// TIA Portal V20 export
FUNCTION_BLOCK "FB_BrakeTest"   // FB412, SCL
TITLE = BrakeTest
{ S7_Optimized_Access := 'FALSE' }
VERSION : 3.12
// Sinamics brake test
// stored: AutoNumber false, IsIECCheckEnabled true, SetENOAutomatically false
   VAR_INPUT
      iStartBt : Bool;   // start BT (Bit must only be resetted as soon as done = 1)
      iQuit : Bool;   // quit error
      iExternalBrakeClosed : Bool;   // feedback external brake; if closed = 1, if open = 0
      iMaxStepTime : Time := T#6S;   // max time per sequencer step
      iBrakeNum : Bool;   // number of brake to be tested; brake 1 = 0; brake 2 = 1
      iActivateAutoDirection : Bool;   // enable automatic detection of direction of test torque
      iSetManualDirection : Bool;   // manual selection of direction of test torque
      iTestSequence : Bool;   // selection of test sequence; sequence 1 = 0, sequence 2 = 1
   END_VAR
   VAR_OUTPUT
      oCloseExternalBrake : Bool;   // signal to close the external brake; close = 1, open = 0
      oDone : Bool;   // done without errors
      oError : Bool;   // error occurred
      oStateNum : Int;   // active step of the sequence
      oDiagnoseError : Int;   // error number
      oError1 : Bool;   // invalid sequence step
      oError2 : Bool;   // invalid start condition: axis not stationery
      oError3 : Bool;   // invalid start condition: pulse enable missing
      oError4 : Bool;   // brake test noch successful
      oError5 : Bool;   // sequence step time monitoring error
      oError6 : Bool;   // startBT reset while in progress
      oError7 : Bool;   // invalid error number
      oError8 : Bool;   // no feedback external brake within "maxStepTime"
   END_VAR
   VAR_IN_OUT
      ioAxisDB : "LBP_typeAxisX";   // UDT of test axis (has to be connected!)
   END_VAR
   VAR
      sStepNum : Int;   // active sequencer step
      sEdgeFlagStop : Bool;   // falling edge flag of startBT
      sEdgeFlagStart : Bool;   // rising edge flag of startBT
      sStepNumOld : Int;   // sequencer step of the previous PLC cycle
      sBTDeselectionDelay : Bool;   // TOF, Q output of deselection timer
      sStartTimer { ExternalVisible := 'False'; ExternalWritable := 'False'} : Bool := true;   // start timer of sequencer time monitoring
      sActiveError : Bool;   // active error
      sInstIecTimerTimeStepBt { S7_SetPoint := 'True'} : TOF_TIME;   // timer for monitoring the steps of the sequencer
      sInstIecTimerSelectSafeBt { S7_SetPoint := 'True'} : TOF_TIME;   // timer to delay the program, if BT is deselected
      sErrorNum { ExternalVisible := 'False'; ExternalWritable := 'False'} : Int;   // provisional error number
   END_VAR
   VAR_TEMP
      tIncrement : Bool;   // increment sequencer
      tTimeSig : Bool;   // TOF, Q output sequencer time monitoring
      tRisBTStart : Bool;   // rising edge startBT
      tFalBTStart : Bool;   // falling edge startBT
      tErr6 : Bool;   // error no. 6
   END_VAR
BEGIN
   REGION BLOCK INFO HEADER
   //=============================================================================
   // Siemens
   // (c)Copyright 2021 All Rights Reserved
   // ----------------------------------------------------------------------------
   // Library:       Lib_SBT_SINUMERIK_ONE
   // Tested with:   V6.13 / NCU 1760
   // Engineering:   TIA Portal V16 Update 4
   // Restrictions:  -
   // Requirements:  motor with brake; UDT "LBP_typeAxisX" of the axis to be tested
   // Functionality: brake test for safety axis
   // ----------------------------------------------------------------------------
   // Change log table:
   // Version   Date         Expert in charge   Changes applied
   // 03.01.02  01.12.2021   Siemens AG         First released version
   // =============================================================================
   END_REGION BLOCK INFO HEADER

   REGION set temp variables 
     #tErr6 := 0;
     #tIncrement := 0;
     #tTimeSig := 0;
     #tRisBTStart := 0;
     #tFalBTStart := 0;
   END_REGION

   REGION edge evaluation 
     // rising edge startBt 
     #tRisBTStart := (#iStartBt AND NOT #iQuit) AND NOT #sEdgeFlagStart;
     #sEdgeFlagStart := (#iStartBt AND NOT #iQuit);

     // falling edge startBt 
     #tFalBTStart := NOT #iStartBt AND #sEdgeFlagStop;
     #sEdgeFlagStop := #iStartBt;
   END_REGION

   REGION return function if Test is inactive 
     // return function while Test is inactive 
     IF NOT (#iStartBt OR #tFalBTStart OR #tRisBTStart OR
       #sActiveError OR #iQuit) THEN
       RETURN;
   END_IF;
   END_REGION

   REGION reset brake test enable when FB stopped 
     IF NOT (#iStartBt OR #sActiveError) THEN
       IF #sStepNum <> 0 THEN
         //error number 6: SBT is cancelled with startBt=0 
         #tErr6 := 1;
       END_IF;
       //stop step sequence 
       #sStepNum := 0;
       //Cancellation/deselection SBT 
       #ioAxisDB.A_StartBrakeTest := 0;
       #ioAxisDB.SCC.CW3.SelectionSBT := 0;
       #ioAxisDB.SCC.CW3.BT_Start := 0;
     END_IF;
   END_REGION

   REGION external brake status/control 
     IF #iStartBt THEN
       //control external brake 
       #oCloseExternalBrake := #ioAxisDB.SIC.SW3.BrakeReq;
       //status external brake 
       #ioAxisDB.SCC.CW3.BrakeClosed := #iExternalBrakeClosed;
     END_IF;

   END_REGION

   REGION timer 
     //start Watchdog Timer on the beginning and for every new step 
     #sStartTimer := 0;
     IF (#sStepNum <> #sStepNumOld)
       OR (#tRisBTStart = 1) THEN
       #sStartTimer := 1;
     END_IF;

     // Timer (TOF) Time delay stop SBT 
     #sInstIecTimerSelectSafeBt(IN := #ioAxisDB.A_StartBrakeTest,
                               PT := T#100ms,
                               Q => #sBTDeselectionDelay);

     // Timer (TOF) Watchdog for step sequence  
     #sInstIecTimerTimeStepBt(IN := #sStartTimer,
                             PT := #iMaxStepTime,
                             Q => #tTimeSig);
     #sStepNumOld := #sStepNum;
   END_REGION

   REGION step sequence 
     //start step sequence with rising Edge startBt 
     IF #tRisBTStart THEN
       #sStepNum := 1;
     END_IF;

     // step sequence Brake test 
     CASE #sStepNum OF
       0:  // step sequence not running 
         #sActiveError := 0;
         #oError := 0;
         #oDone := 0;
         #sErrorNum := 0;
       1:  // Check start condition 
         IF NOT #ioAxisDB.E_Stat THEN
           //Axis/spindle is not stationary(n < nmin) 
           //Error Number 2 
           #sErrorNum := 2;
         END_IF;
         IF NOT #ioAxisDB.E_PulseEnable OR NOT #ioAxisDB.E_DriveRunEn THEN
           //Pulse or controller enable is missing 
           //Error Number 3 
           #sErrorNum := 3;
         END_IF;
         IF (#sErrorNum = 0) AND #tTimeSig THEN
           #tIncrement := 1; //next Step                     
         END_IF;

       2:  //Select Brake 1 OR 2 
         #ioAxisDB.SCC.CW3.Brake_1_2 := #iBrakeNum;
         IF #tTimeSig = 1 THEN
           #tIncrement := 1;//next Step  
         END_IF;

       3:  //Select Test sequence 1 or 2 
         #ioAxisDB.SCC.CW3.Testseq_1_2 := #iTestSequence;
         IF #tTimeSig = 1 THEN
           #tIncrement := 1;//next Step  
         END_IF;

       4:  //Set NCK Start signal for Brake test 
         #ioAxisDB.A_StartBrakeTest := 1;
         //feedback NCK Brake test active #axisDB.E_BrakeTest 
         IF (#ioAxisDB.E_BrakeTest) AND (#tTimeSig) THEN
           #tIncrement := 1;//next Step  
         END_IF;

       5:  // Select SBT  
         #ioAxisDB.SCC.CW3.SelectionSBT := 1;
         //feedback SBT selected #axisDB.SIC.SW3.SBT_Sel and test torque from drive #axisDB.SIC.SW3.SetpSettingDrive 
         IF (#tTimeSig = 1) AND #ioAxisDB.SIC.SW3.SBT_Sel AND #ioAxisDB.SIC.SW3.SetpSettingDrive THEN
           #tIncrement := 1;//next Step  
         END_IF;
       6: //Select manual or auto direction  
         IF #iActivateAutoDirection = 1 THEN
           //auto direction 
           #ioAxisDB.SCC.CW3.DirOfROT := #ioAxisDB.SIC.SW3.SignLoadTorque;
         ELSE
           //Manual direction  
           // #setManualDirection=false negative direction 
           // #setManualDirection=true positive direction 
           #ioAxisDB.SCC.CW3.DirOfROT := #iSetManualDirection;
         END_IF;

         IF #tTimeSig = 1 THEN
           #tIncrement := 1;//next Step  
         END_IF;

       7:  // Request start Brake test SCC 
         #ioAxisDB.SCC.CW3.BT_Start := 1;
         //feedback Brake test active SIC #axisDB.SIC.SW3.BT_Act 
         IF #ioAxisDB.SIC.SW3.BT_Act AND #tTimeSig THEN
           #tIncrement := 1;//next Step  
         END_IF;
       8: //Check if the condition of the external brake fits the request 
         IF ((#ioAxisDB.SIC.SW3.BrakeReq XOR #ioAxisDB.SCC.CW3.BrakeClosed) AND (NOT #tTimeSig)) THEN
           //Error external Brake 
           #sErrorNum := 8;
         END_IF;

         IF (#ioAxisDB.SIC.SW3.BrakeReq = #ioAxisDB.SCC.CW3.BrakeClosed) AND #tTimeSig THEN

           #tIncrement := 1;//next Step  
         END_IF;

       9:  // Waiting for SBT finished signal 
         IF #ioAxisDB.SIC.SW3.BT_Finished AND #tTimeSig THEN
           #tIncrement := 1;//next Step  
         END_IF;
       10: // Check if SBT was OK 
         IF NOT (#ioAxisDB.SIC.SW3.BT_Finished AND #ioAxisDB.SIC.SW3.BT_OK) THEN
           //SBT finished with error 
           #sErrorNum := 4;
         END_IF;
         IF #tTimeSig AND #ioAxisDB.SIC.SW3.BT_OK THEN
           #tIncrement := 1;//next Step  
         END_IF;
       11: // Request stop Brake test SCC 
         #ioAxisDB.SCC.CW3.BT_Start := 0;
         IF #tTimeSig AND NOT (#ioAxisDB.SIC.SW3.BT_Act AND #sBTDeselectionDelay) THEN
           //Feedback SIC SBT is stopped  
           #tIncrement := 1;//next Step  
         END_IF;
       12: // Reset NCK Start signal for Brake test 
         // Deselect SBT via SCC 
         #ioAxisDB.A_StartBrakeTest := 0;
         #ioAxisDB.SCC.CW3.SelectionSBT := 0;
         IF #tTimeSig AND NOT #ioAxisDB.E_BrakeTest AND NOT #ioAxisDB.SIC.SW3.SBT_Sel THEN
           // SBT finished without error 
           // set done 
           // stop step sequence 
           #sStepNum := 0;
           #oDone := 1;
         END_IF;
       ELSE:
         //wrong step number 
         #sErrorNum := 1;
   END_CASE;
   END_REGION

   REGION error handling 
     // error number 6: SBT is cancelled with startBt=0 while running without error 
     IF #tErr6 THEN
       //Error Number 6 
       #sErrorNum := 6;
       //set error 
       #oError := 1;
     END_IF;

     // Watchdog step sequence -> Error Num 5 
     IF #sErrorNum = 0 AND (#sStepNum <> 0) AND NOT #tTimeSig THEN
       #sErrorNum := 5;
       #oError := 1;
       #sActiveError := 1;
     END_IF;

     // Error Bit 
     CASE #sErrorNum OF
       0:
         ;
       1:
         #oError1 := 1;
       2:
         #oError2 := 1;
       3:
         #oError3 := 1;
       4:
         #oError4 := 1;
       5:
         #oError5 := 1;
       6:
         #oError6 := 1;
       8:
         #oError8 := 1;
       ELSE                  // Wrong error number -> set Error Num 7
         #oError7 := 1;
         #sErrorNum := 7;
     END_CASE;

     // output error number and step number for diagnose 
     IF #sErrorNum <> 0 THEN
         #oError := 1;
         #sActiveError := 1;
         #oDiagnoseError := #sErrorNum;
         #oStateNum := #sStepNum;
     END_IF;
   END_REGION

   REGION quit error 
     //reset signals  
       IF #iQuit = 1 THEN
           #ioAxisDB.SCC.CW3.BT_Start := 0;
           #ioAxisDB.A_StartBrakeTest := 0;
           #ioAxisDB.SCC.CW3.Brake_1_2 := 0;
           #ioAxisDB.SCC.CW3.SelectionSBT := 0;
           #oCloseExternalBrake := 0;
           #sStartTimer := 1;
           #oError := 0;
           #oError1 := 0;
           #oError2 := 0;
           #oError3 := 0;
           #oError4 := 0;
           #oError5 := 0;
           #oError6 := 0;
           #oError7 := 0;
           #oError8 := 0;
           #sActiveError := 0;
           #oDiagnoseError := 0;
           #oStateNum := 0;
           #sStepNum := 0;
           #tIncrement := 0;
       END_IF;
   END_REGION

   REGION increment step sequence 
     //increment step number 
     IF #sErrorNum = 0 AND #tIncrement = 1 THEN
       //increment step number 
       #sStepNum += 1;
       //update output step number 
       #oStateNum := #sStepNum;
   END_IF;
   END_REGION
END_FUNCTION_BLOCK
